// TIA Portal V20 export
DATA_BLOCK "DB_PowermeterMeasures"   // DB434
TITLE = DB_MEAS_POWER_METER
{ S7_Optimized_Access := 'TRUE' }
AUTHOR : SAN
// Measures of power metter
// stored: AutoNumber false, InstanceOfName UDT_PowermeterMeasure, InstanceOfType UDT
"UDT_PowermeterMeasure"
   // VAR RETAIN
   //    NbMeasure : Int;
   //    ActualMeasure : Int;
   //    ActualTotalMeas : Real;
   //    Table_full : Bool;
   //    Measures : Array[0..99] of Struct
   //       Time_day : Time_Of_Day;
   //       Day_meas : Date;
   //       Job_meas : Int;
   //       ValuePower : Real;
   //       ValueCM : Real;
   //    END_STRUCT;
   // END_VAR
BEGIN
END_DATA_BLOCK
